// TIA Portal project "G120 Shoxrux" (V15.1)

(* hardware
DEVICE "S71500/ET200MP station_1"  S7-1500 station
   slot 0: "Rail_0"  Rack  6ES7 590-1***0-0AA0
   slot 1: "I am a brain"  CPU 1511C-1 PN  6ES7 511-1CK00-0AB0  V2.6
      slot 3: "CPU display_1"  6ES7591-1AA00-0AA0
DEVICE "SINAMICS G_1"  Sinamics.Device
   slot 0: "	_0"  Rail  SinamicsG120RackPN
   slot 0: "I am a driver"  G120 CU240E-2 PN-F  6SL3244-0BB13-1FA0  4.7.10
      slot 1: "PROFINET interface"  MDD-SinamicsG120-P
   slot 3: "PM240 IP20"  PM240 IP20  6SL3224-0BE13-7UA0  -
*)

// ===== PLC "I am a brain"  CPU 1511C-1 PN =====

VAR_GLOBAL   // PLC tag table "Default tag table"
   "Tag_1" AT %IW20 : Word;
   "Tag_2" AT %M0.0 : Bool;
END_VAR

VAR_GLOBAL   // PLC tag table "Motor Data"
   "Motor SetPoin speed" AT %QW258 : Int;
   "Motor potesiometr" AT %MW40 : Int;
   "Normalized Speed" AT %MD42 : Real;
   "Cleareance_0" AT %Q256.2 : Bool;
   "Cleareance_1" AT %Q257.1 : Bool;
   "Cleareance_2" AT %Q257.2 : Bool;
   "Cleareance_3" AT %Q257.3 : Bool;
   "Cleareance_4" AT %Q257.4 : Bool;
   "Cleareance_5" AT %Q257.5 : Bool;
   "Cleareance_6" AT %Q257.6 : Bool;
   "Cleareance_7" AT %Q257.7 : Bool;
   "Motor ON" AT %Q257.0 : Bool;
   "Motor ON push button" AT %I0.2 : Bool;
   "Motor Reverse Switch" AT %I0.3 : Bool;
   "Motor Reverse" AT %Q256.3 : Bool;
END_VAR

FUNCTION "Motor" : Void   // FC1, LAD
{ S7_Optimized_Access := 'TRUE' }
VERSION : 0.1
BEGIN

REGION Network 1
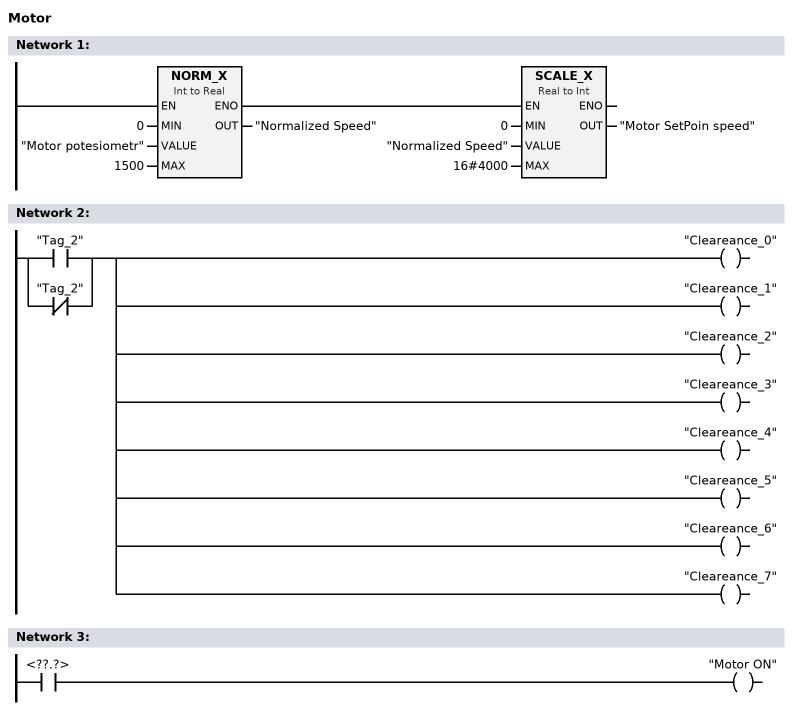
   RUNG wire#powerrail
      { S7_Templates := "[SrcType := Int, DestType := Real]" } Normalize(min := 0, value := "Motor potesiometr", max := 1500, out => "Normalized Speed")
      { S7_Templates := "[SrcType := Real, DestType := Int]" } Scale(min := 0, value := "Normalized Speed", max := 16#4000, out => "Motor SetPoin speed")
   END_RUNG
   // the same network as SCL:
   "Normalized Speed" := NORM_X(MIN := 0, VALUE := "Motor potesiometr", MAX := 1500);
   "Motor SetPoin speed" := SCALE_X(MIN := 0, VALUE := "Normalized Speed", MAX := 16#4000);
END_REGION

REGION Network 2
   RUNG wire#powerrail
      Contact( "Tag_2" )
      wire#w1
      Coil( "Cleareance_0" )
   END_RUNG
   RUNG wire#powerrail
      I_Contact( "Tag_2" )
   END_RUNG wire#w1
   RUNG wire#w1
      Coil( "Cleareance_1" )
   END_RUNG
   RUNG wire#w1
      Coil( "Cleareance_2" )
   END_RUNG
   RUNG wire#w1
      Coil( "Cleareance_3" )
   END_RUNG
   RUNG wire#w1
      Coil( "Cleareance_4" )
   END_RUNG
   RUNG wire#w1
      Coil( "Cleareance_5" )
   END_RUNG
   RUNG wire#w1
      Coil( "Cleareance_6" )
   END_RUNG
   RUNG wire#w1
      Coil( "Cleareance_7" )
   END_RUNG
   // the same network as SCL:
   "Cleareance_0" := "Tag_2" OR NOT "Tag_2";
   "Cleareance_1" := "Cleareance_0";
   "Cleareance_2" := "Cleareance_0";
   "Cleareance_3" := "Cleareance_0";
   "Cleareance_4" := "Cleareance_0";
   "Cleareance_5" := "Cleareance_0";
   "Cleareance_6" := "Cleareance_0";
   "Cleareance_7" := "Cleareance_0";
END_REGION

REGION Network 3
   RUNG wire#powerrail
      Contact(  )
      Coil( "Motor ON" )
   END_RUNG
   // the same network as SCL:
   // no checked SCL form for this network; see the picture
END_REGION
END_FUNCTION

ORGANIZATION_BLOCK "Main"   // OB1, LAD, ProgramCycle
TITLE = "Main Program Sweep (Cycle)"
{ S7_Optimized_Access := 'TRUE' }
VERSION : 0.1
   VAR_INPUT
      Initial_Call : Bool;   // Initial call of this OB
      Remanence : Bool;   // =True, if remanent data are available
   END_VAR
BEGIN

REGION Network 1
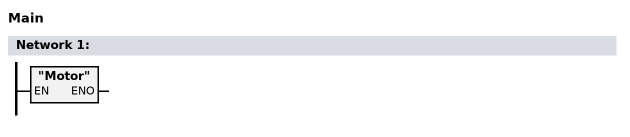
   RUNG wire#powerrail
      "Motor"()
   END_RUNG
   // the same network as SCL:
   "Motor"();
END_REGION
END_ORGANIZATION_BLOCK